// TIA Portal V20 export
DATA_BLOCK "T5 EXCENTRIC PARAMETERS"   // DB1318
{ S7_Optimized_Access := 'TRUE' }
// stored: AutoNumber false, MemoryReserve 100
   VAR RETAIN
      "-" : Int;
   END_VAR
BEGIN
END_DATA_BLOCK
